// TIA Portal V19 export
TYPE "LEXCHANGETRAY_typePlasticEm5_toHandlingXyzDeliver"
// stored: Access Published
   STRUCT
      req : "LEXCHANGETRAY_typePlasticEm5_toHandlingXyzReq";
      feedback { S7_SetPoint := 'True'} : "LEXCHANGETRAY_typePlasticEm5_toHandlingXyzFeedback";
   END_STRUCT;
END_TYPE
